FUNCTION_BLOCK PUBLIC FB_Base
VAR_INPUT
END_VAR
VAR_OUTPUT
END_VAR
VAR
END_VAR

END_FUNCTION_BLOCK

(* stored: Version 1.1.0.1, ProductVersion 3.1.4022.10
   POU FB_Base: Id {d1bd9f66-ea51-4f58-97c6-de9ed5be3541}, SpecialFunc None *)
